SYSTEM FBTypeDeleteNestedSubAppTest
  (* Version 1.0, 2026-06-15, Dimitrios Kalligaridis *)
  APPLICATION App
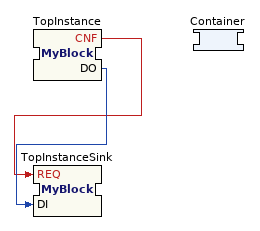
    FBS
      TopInstance : mypackage::MyBlock;
      TopInstanceSink : mypackage::MyBlock;
    END_FBS
    SUBAPPLICATION Container
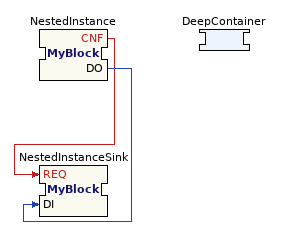
      FBS
        NestedInstance : mypackage::MyBlock;
        NestedInstanceSink : mypackage::MyBlock;
      END_FBS
      SUBAPPLICATION DeepContainer
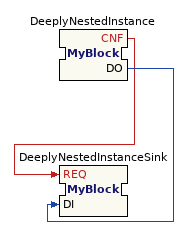
        FBS
          DeeplyNestedInstance : mypackage::MyBlock;
          DeeplyNestedInstanceSink : mypackage::MyBlock;
        END_FBS
        EVENT_CONNECTIONS
          DeeplyNestedInstance.CNF TO DeeplyNestedInstanceSink.REQ;
        END_CONNECTIONS
        DATA_CONNECTIONS
          DeeplyNestedInstance.DO TO DeeplyNestedInstanceSink.DI;
        END_CONNECTIONS
      END_SUBAPPLICATION
      EVENT_CONNECTIONS
        NestedInstance.CNF TO NestedInstanceSink.REQ;
      END_CONNECTIONS
      DATA_CONNECTIONS
        NestedInstance.DO TO NestedInstanceSink.DI;
      END_CONNECTIONS
    END_SUBAPPLICATION
    EVENT_CONNECTIONS
      TopInstance.CNF TO TopInstanceSink.REQ;
    END_CONNECTIONS
    DATA_CONNECTIONS
      TopInstance.DO TO TopInstanceSink.DI;
    END_CONNECTIONS
  END_APPLICATION
END_SYSTEM
